// TIA Portal V20 export
VAR_GLOBAL   // PLC tag table "unit_status"
END_VAR
VAR_GLOBAL CONSTANT   // user constants
   NOT_DEFINED : DInt := 0;
   EMPTY : DInt := 2;
   WORKING : DInt := 3;
   RAW : DInt := 4;
   FINISHED : DInt := 5;
   PAUSED : DInt := 6;
   ABORTED : DInt := 7;
   LOCKED : DInt := 9;
   AUTO : DInt := 10;   // nonUsare
   MANUAL : DInt := 20;   // nonUsare
   ALARM : DInt := 99;
   LOADED : DInt := 1;
   UNLOADED : DInt := 100;   // totally empty machine
   OFF : DInt := 999;
   HOLD : DInt := 17;
   REMOTE : DInt := 15;
   _LOCAL : DInt := 16;
   READY_TO_WORK : DInt := 12;
   WAITING_MATERIAL : DInt := 13;
END_VAR
